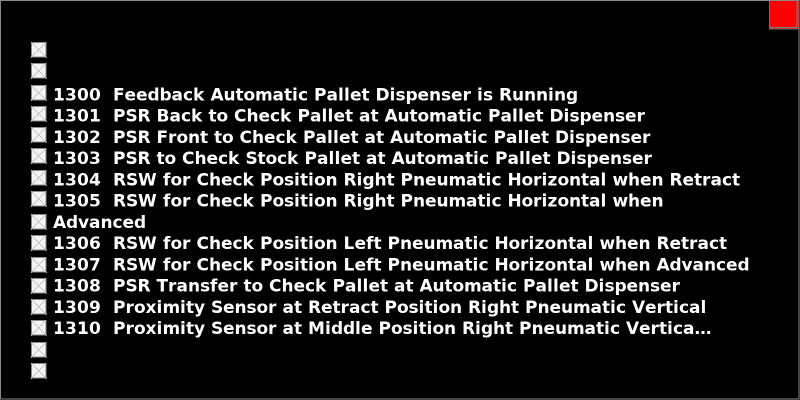
VISUALIZATION P2_DI4  // 800x400, background image 
    ImageSwitcher (31,42 15x15), variable: InputOutput_GVL.Digital_Input[49], behaviour: TOGGLE
    Label (50,16 705x391), "1300 Feedback Automatic Pallet Dispenser is Running 1301 PSR Back to Check Pallet at Automatic Pallet Dispenser 1302 PSR Front to Check Pallet at Automatic Pallet Dispenser 1303 PSR to Check Stock Pallet at Automatic Pallet Dispenser 1304 RSW for Check Position Right Pneumatic Horizontal when Retract 1305 RSW for Check Position Right Pneumatic Horizontal when Advanced 1306 RSW for Check Position Left Pneumatic Horizontal when Retract 1307 RSW for Check Position Left Pneumatic Horizontal when Advanced 1308 PSR Transfer to Check Pallet at Automatic Pallet Dispenser 1309 Proximity Sensor at Retract Position Right Pneumatic Vertical 1310 Proximity Sensor at Middle Position Right Pneumatic Vertical 1311 Proximity Sensor at Advanced Position Right Pneumatic Vertical 1312 Proximity Sensor at Retract Position Left Pneumatic Vertical 1313 Proximity Sensor at Middle Position Left Pneumatic Vertical 1314 Proximity Sensor at Advanced Position Left Pneumatic Vertical 1315 Request Release Solenoid Door Outfeed"
    ImageSwitcher (31,63 15x15), variable: InputOutput_GVL.Digital_Input[50], behaviour: TOGGLE
    ImageSwitcher (31,85 15x15), variable: InputOutput_GVL.Digital_Input[51], behaviour: TOGGLE
    ImageSwitcher (31,106 15x15), variable: InputOutput_GVL.Digital_Input[52], behaviour: TOGGLE
    ImageSwitcher (31,127 15x15), variable: InputOutput_GVL.Digital_Input[53], behaviour: TOGGLE
    ImageSwitcher (31,148 15x15), variable: InputOutput_GVL.Digital_Input[54], behaviour: TOGGLE
    ImageSwitcher (31,170 15x15), variable: InputOutput_GVL.Digital_Input[55], behaviour: TOGGLE
    ImageSwitcher (31,191 15x15), variable: InputOutput_GVL.Digital_Input[56], behaviour: TOGGLE
    ImageSwitcher (31,214 15x15), variable: InputOutput_GVL.Digital_Input[57], behaviour: TOGGLE
    ImageSwitcher (31,235 15x15), variable: InputOutput_GVL.Digital_Input[58], behaviour: TOGGLE
    ImageSwitcher (31,257 15x15), variable: InputOutput_GVL.Digital_Input[59], behaviour: TOGGLE
    ImageSwitcher (31,278 15x15), variable: InputOutput_GVL.Digital_Input[60], behaviour: TOGGLE
    ImageSwitcher (31,299 15x15), variable: InputOutput_GVL.Digital_Input[61], behaviour: TOGGLE
    ImageSwitcher (31,320 15x15), variable: InputOutput_GVL.Digital_Input[62], behaviour: TOGGLE
    ImageSwitcher (31,342 15x15), variable: InputOutput_GVL.Digital_Input[63], behaviour: TOGGLE
    ImageSwitcher (31,363 15x15), variable: InputOutput_GVL.Digital_Input[64], behaviour: TOGGLE
    Button (769,-1 30x30), image: VisuSymbols.Symbols.Wrong
        OnMouseClick: CloseDialog Dialog=P2_DI4, Result=OK, NumpadKeypadSet=True
END_VISUALIZATION

(* stored: Version 1.1.0.1, ProductVersion 3.1.4024.12
   Visu P2_DI4: Id {5fdfd043-0dcb-44ac-b4e5-ee6c04e36fea} *)
